Fanuc KAREL source: kb00151.KL

-- PROVISIONAL review KL for V1013-1; original PC SHA256 455141145e3ebcaac28aae7cf142150b6b9a4ed6ff4c94258d204909a9e5fae4
-- Incomplete behavior may be omitted. Consult companion uncertainty JSON. Do not deploy.
PROGRAM KB00151
%NOLOCKGROUP
BEGIN
  -- UNRESOLVED_PC offsets 5-14; opcodes 3F,75
  -- UNRESOLVED_PC offsets 19-26; opcodes 9D,23
  -- UNRESOLVED_PC offsets 31-38; opcodes 9D,23
  -- UNRESOLVED_PC offsets 43-73; opcodes 27,22,2A,22,22,22,31
  -- UNRESOLVED_PC offsets 78-82; opcodes 7F
END KB00151
